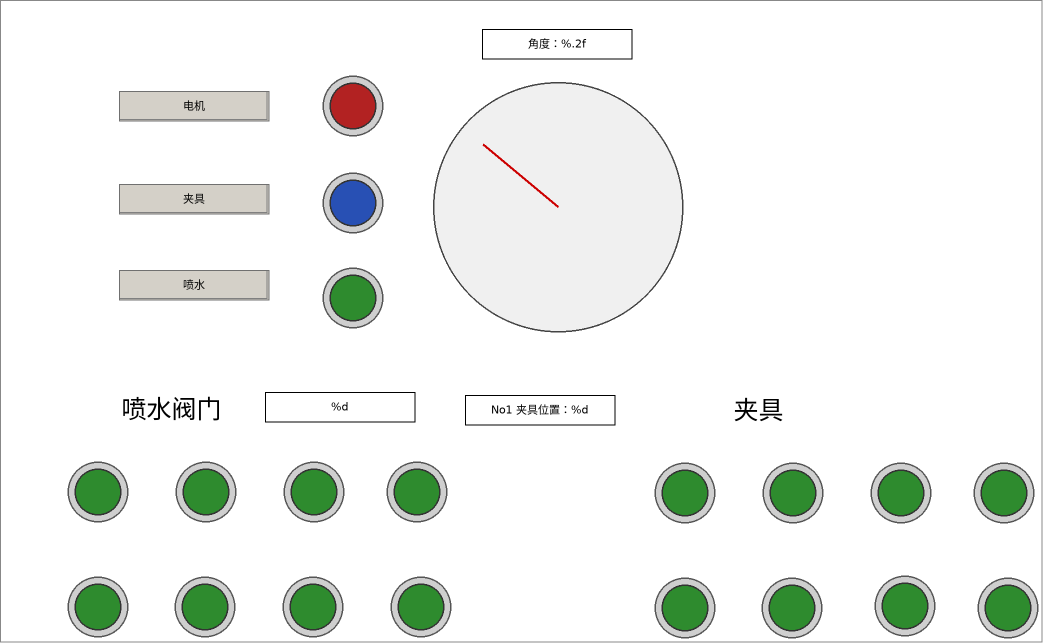
VISUALIZATION Visualization  // 1043x643
    Button (119,91 150x30), "电机"
        OnMouseClick: execute { MAIN.ServoDo :=NOT MAIN.ServoDo; }
    Meter360 (433,82 250x250), value: MAIN.Controller.CurrentAngle, style: Meter-Meter360-Red, scale format: %.1f, scale 0..360
    Button (119,270 150x30), "喷水"
        OnMouseClick: execute { MAIN.SprayExecute:= NOT MAIN.SprayExecute; }
    Button (119,184 150x30), "夹具"
        OnMouseClick: execute { MAIN.FixtureEnable:= NOT MAIN.FixtureEnable; }
    Lamp1 (318,71 70x70), variable: MAIN.ServoDo, style: Lamp-Lamp1-Red
    Lamp1 (318,168 70x70), variable: MAIN.FixtureEnable, style: Lamp-Lamp1-Blue
    Lamp1 (318,263 70x70), variable: MAIN.SprayExecute, style: Lamp-Lamp1-Green
    Lamp1 (63,457 70x70), variable: MAIN.spray.SpraySwitch[0], style: Lamp-Lamp1-Green
    Lamp1 (171,457 70x70), variable: MAIN.spray.SpraySwitch[1], style: Lamp-Lamp1-Green
    Lamp1 (279,457 70x70), variable: MAIN.spray.SpraySwitch[2], style: Lamp-Lamp1-Green
    Lamp1 (382,457 70x70), variable: MAIN.spray.SpraySwitch[3], style: Lamp-Lamp1-Green
    Lamp1 (63,572 70x70), variable: MAIN.spray.SpraySwitch[4], style: Lamp-Lamp1-Green
    Lamp1 (170,572 70x70), variable: MAIN.spray.SpraySwitch[5], style: Lamp-Lamp1-Green
    Lamp1 (278,572 70x70), variable: MAIN.spray.SpraySwitch[6], style: Lamp-Lamp1-Green
    Lamp1 (386,572 70x70), variable: MAIN.spray.SpraySwitch[7], style: Lamp-Lamp1-Green
    Label (65,390 213x38), "喷水阀门"
    Rectangle (482,29 150x30), "角度：%.2f", text variable: MAIN.Controller.CurrentAngle
    Rectangle (265,392 150x30), "%d", text variable: MAIN.spray.Order[2]
    Rectangle (465,395 150x30), "No1 夹具位置：%d", text variable: MAIN.spray.pick+1
    Lamp1 (650,458 70x70), variable: MAIN.FixtureStateArray[0], style: Lamp-Lamp1-Green
    Lamp1 (758,458 70x70), variable: MAIN.FixtureStateArray[1], style: Lamp-Lamp1-Green
    Lamp1 (866,458 70x70), variable: MAIN.FixtureStateArray[2], style: Lamp-Lamp1-Green
    Lamp1 (969,458 70x70), variable: MAIN.FixtureStateArray[3], style: Lamp-Lamp1-Green
    Lamp1 (650,573 70x70), variable: MAIN.FixtureStateArray[4], style: Lamp-Lamp1-Green
    Lamp1 (757,573 70x70), variable: MAIN.FixtureStateArray[5], style: Lamp-Lamp1-Green
    Lamp1 (870,571 70x70), variable: MAIN.FixtureStateArray[6], style: Lamp-Lamp1-Green
    Lamp1 (973,573 70x70), variable: MAIN.FixtureStateArray[7], style: Lamp-Lamp1-Green
    Label (652,391 213x38), "夹具"
END_VISUALIZATION

(* stored: Version 1.1.0.1, ProductVersion 3.1.4024.12
   Visu Visualization: Id {47d50a6f-f1c1-4cd6-a2a9-61b9d81c9eca} *)
